// TIA Portal V20 export
DATA_BLOCK "Instance_FB_IO_Device_DB"   // DB104
// stored: AutoNumber false, InstanceOfName FB_IO_Device, InstanceOfType FB
"FB_IO_Device"
   // VAR_INPUT
   //    Test_Station : SInt;
   //    Life_Trigger : Bool;
   //    Star_Test : Bool;
   //    Button_Start_Approve : Bool;
   //    Electrical_Current_Test_Approved : Bool;
   //    Visual_Test_Approved : Bool;
   //    Electrical_Current_Read : UInt;
   //    In_Functional_Test : "IO_Device_Functinal_Test";
   //    In_Test_Parameters : "IO_Device_Test_Parameters";
   // END_VAR
   // VAR_OUTPUT
   //    Reset_Functional_Test : Bool;
   //    Out_Test_Parameters : "IO_Device_Test_Parameters";
   //    Out_Functional_Test : "IO_Device_Functinal_Test";
   // END_VAR
BEGIN
END_DATA_BLOCK
